// Mitsubishi GX Works2 project: maykhoai   PLC: FX3U/FX3UC

// global labels: Global1
VAR_GLOBAL
  DC AT Y000 : BOOL;
  HH AT Y001 : BOOL;
  XL_CK AT Y002 : BOOL;
  DAU AT Y003 : BOOL;
  SS_CUT AT X000 : BOOL;
END_VAR

PROGRAM MAIN
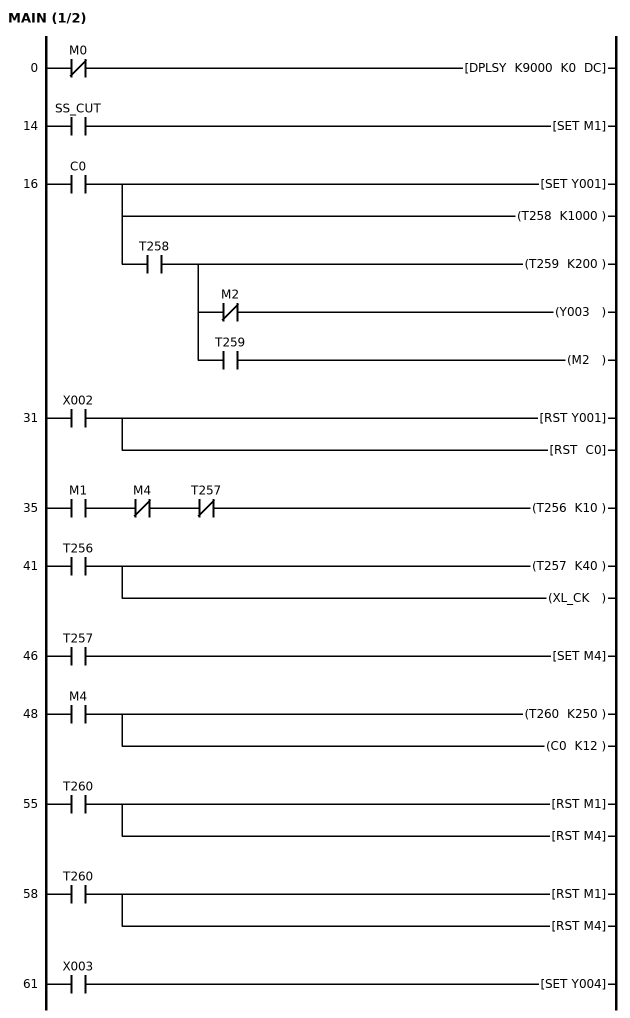
0     LDI     M0
      DPLSY   K9000 K0 DC
14    LD      SS_CUT
      SET     M1
16    LD      C0
      SET     Y001
      OUT     T258 K1000
      AND     T258
      OUT     T259 K200
      MPS
      ANI     M2
      OUT     Y003
      MPP
      AND     T259
      OUT     M2
31    LD      X002
      RST     Y001
      RST     C0
35    LD      M1
      ANI     M4
      ANI     T257
      OUT     T256 K10
41    LD      T256
      OUT     T257 K40
      OUT     XL_CK
46    LD      T257
      SET     M4
48    LD      M4
      OUT     T260 K250
      OUT     C0 K12
55    LD      T260
      RST     M1
      RST     M4
58    LD      T260
      RST     M1
      RST     M4
61    LD      X003
      SET     Y004
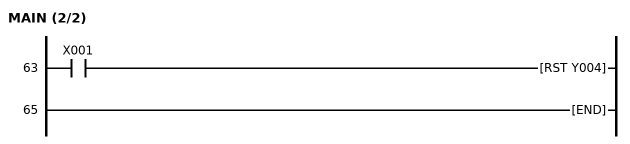
63    LD      X001
      RST     Y004
65    END
END_PROGRAM
